// Mitsubishi GX Developer project: パレット取り外し   PLC: Q02

PROGRAM ALARM
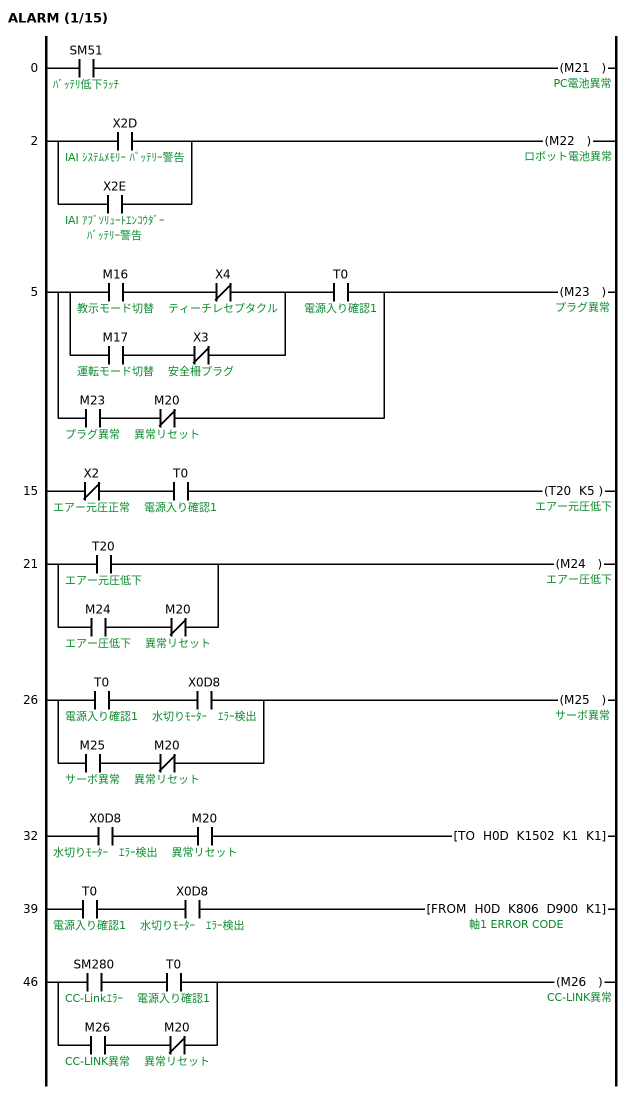
0     LD      SM51  ; ﾊﾞｯﾃﾘ低下ﾗｯﾁ
      OUT     M21  ; PC電池異常
2     LD      X2D  ; IAI ｼｽﾃﾑﾒﾓﾘｰ ﾊﾞｯﾃﾘｰ警告
      OR      X2E  ; IAI ｱﾌﾞｿﾘｭｰﾄｴﾝｺｳﾀﾞｰ ﾊﾞｯﾃﾘｰ警告
      OUT     M22  ; ロボット電池異常
5     LD      M16  ; 教示モード切替
      ANI     X4  ; ティーチレセプタクル
      LD      M17  ; 運転モード切替
      ANI     X3  ; 安全柵プラグ
      ORB
      AND     T0  ; 電源入り確認1
      LD      M23  ; プラグ異常
      ANI     M20  ; 異常リセット
      ORB
      OUT     M23  ; プラグ異常
15    LDI     X2  ; エアー元圧正常
      AND     T0  ; 電源入り確認1
      OUT     T20 K5  ; エアー元圧低下
21    LD      T20  ; エアー元圧低下
      LD      M24  ; エアー圧低下
      ANI     M20  ; 異常リセット
      ORB
      OUT     M24  ; エアー圧低下
26    LD      T0  ; 電源入り確認1
      AND     X0D8  ; 水切りﾓｰﾀｰ　ｴﾗｰ検出
      LD      M25  ; サーボ異常
      ANI     M20  ; 異常リセット
      ORB
      OUT     M25  ; サーボ異常
32    LD      X0D8  ; 水切りﾓｰﾀｰ　ｴﾗｰ検出
      AND     M20  ; 異常リセット
      TO      H0D K1502 K1 K1
39    LD      T0  ; 電源入り確認1
      AND     X0D8  ; 水切りﾓｰﾀｰ　ｴﾗｰ検出
      FROM    H0D K806 D900 K1  ; 軸1 ERROR CODE
46    LD      SM280  ; CC-Linkｴﾗｰ
      AND     T0  ; 電源入り確認1
      LD      M26  ; CC-LINK異常
      ANI     M20  ; 異常リセット
      ORB
      OUT     M26  ; CC-LINK異常
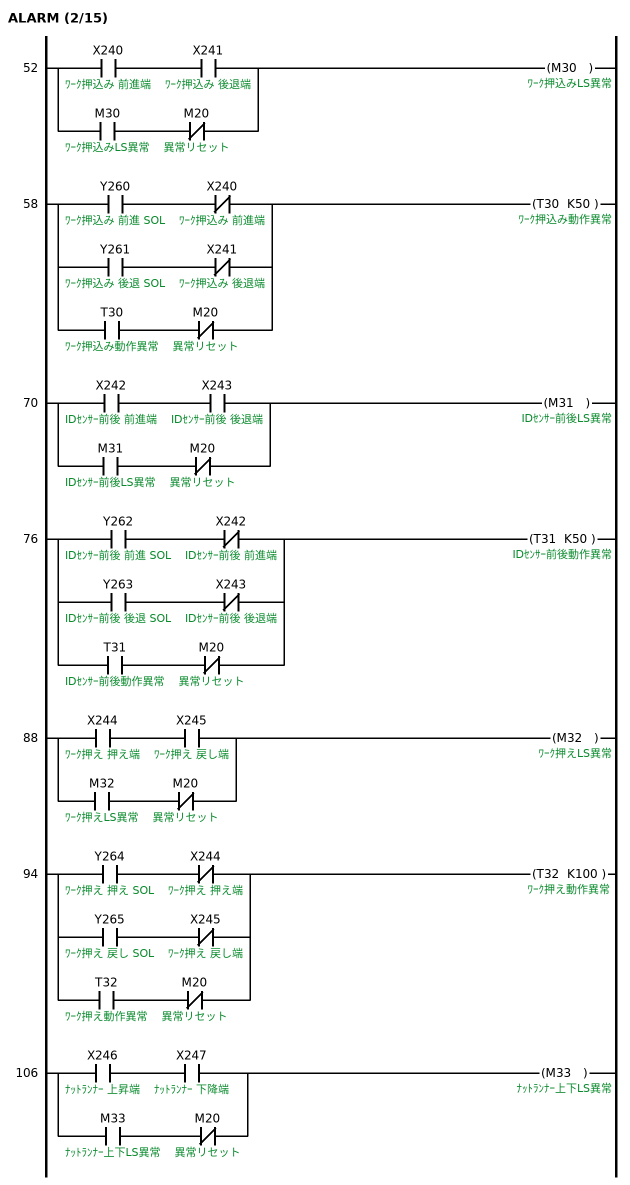
52    LD      X240  ; ﾜｰｸ押込み 前進端
      AND     X241  ; ﾜｰｸ押込み 後退端
      LD      M30  ; ﾜｰｸ押込みLS異常
      ANI     M20  ; 異常リセット
      ORB
      OUT     M30  ; ﾜｰｸ押込みLS異常
58    LD      Y260  ; ﾜｰｸ押込み 前進 SOL
      ANI     X240  ; ﾜｰｸ押込み 前進端
      LD      Y261  ; ﾜｰｸ押込み 後退 SOL
      ANI     X241  ; ﾜｰｸ押込み 後退端
      ORB
      LD      T30  ; ﾜｰｸ押込み動作異常
      ANI     M20  ; 異常リセット
      ORB
      OUT     T30 K50  ; ﾜｰｸ押込み動作異常
70    LD      X242  ; IDｾﾝｻｰ前後 前進端
      AND     X243  ; IDｾﾝｻｰ前後 後退端
      LD      M31  ; IDｾﾝｻｰ前後LS異常
      ANI     M20  ; 異常リセット
      ORB
      OUT     M31  ; IDｾﾝｻｰ前後LS異常
76    LD      Y262  ; IDｾﾝｻｰ前後 前進 SOL
      ANI     X242  ; IDｾﾝｻｰ前後 前進端
      LD      Y263  ; IDｾﾝｻｰ前後 後退 SOL
      ANI     X243  ; IDｾﾝｻｰ前後 後退端
      ORB
      LD      T31  ; IDｾﾝｻｰ前後動作異常
      ANI     M20  ; 異常リセット
      ORB
      OUT     T31 K50  ; IDｾﾝｻｰ前後動作異常
88    LD      X244  ; ﾜｰｸ押え 押え端
      AND     X245  ; ﾜｰｸ押え 戻し端
      LD      M32  ; ﾜｰｸ押えLS異常
      ANI     M20  ; 異常リセット
      ORB
      OUT     M32  ; ﾜｰｸ押えLS異常
94    LD      Y264  ; ﾜｰｸ押え 押え SOL
      ANI     X244  ; ﾜｰｸ押え 押え端
      LD      Y265  ; ﾜｰｸ押え 戻し SOL
      ANI     X245  ; ﾜｰｸ押え 戻し端
      ORB
      LD      T32  ; ﾜｰｸ押え動作異常
      ANI     M20  ; 異常リセット
      ORB
      OUT     T32 K100  ; ﾜｰｸ押え動作異常
106   LD      X246  ; ﾅｯﾄﾗﾝﾅｰ 上昇端
      AND     X247  ; ﾅｯﾄﾗﾝﾅｰ 下降端
      LD      M33  ; ﾅｯﾄﾗﾝﾅｰ上下LS異常
      ANI     M20  ; 異常リセット
      ORB
      OUT     M33  ; ﾅｯﾄﾗﾝﾅｰ上下LS異常
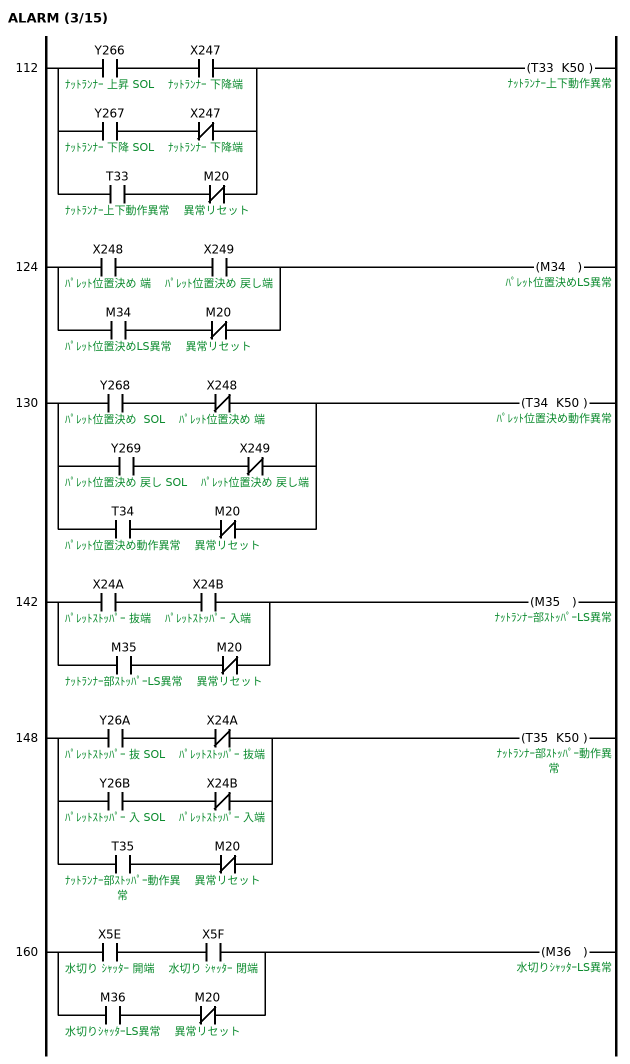
112   LD      Y266  ; ﾅｯﾄﾗﾝﾅｰ 上昇 SOL
      AND     X247  ; ﾅｯﾄﾗﾝﾅｰ 下降端
      LD      Y267  ; ﾅｯﾄﾗﾝﾅｰ 下降 SOL
      ANI     X247  ; ﾅｯﾄﾗﾝﾅｰ 下降端
      ORB
      LD      T33  ; ﾅｯﾄﾗﾝﾅｰ上下動作異常
      ANI     M20  ; 異常リセット
      ORB
      OUT     T33 K50  ; ﾅｯﾄﾗﾝﾅｰ上下動作異常
124   LD      X248  ; ﾊﾟﾚｯﾄ位置決め 端
      AND     X249  ; ﾊﾟﾚｯﾄ位置決め 戻し端
      LD      M34  ; ﾊﾟﾚｯﾄ位置決めLS異常
      ANI     M20  ; 異常リセット
      ORB
      OUT     M34  ; ﾊﾟﾚｯﾄ位置決めLS異常
130   LD      Y268  ; ﾊﾟﾚｯﾄ位置決め  SOL
      ANI     X248  ; ﾊﾟﾚｯﾄ位置決め 端
      LD      Y269  ; ﾊﾟﾚｯﾄ位置決め 戻し SOL
      ANI     X249  ; ﾊﾟﾚｯﾄ位置決め 戻し端
      ORB
      LD      T34  ; ﾊﾟﾚｯﾄ位置決め動作異常
      ANI     M20  ; 異常リセット
      ORB
      OUT     T34 K50  ; ﾊﾟﾚｯﾄ位置決め動作異常
142   LD      X24A  ; ﾊﾟﾚｯﾄｽﾄｯﾊﾟｰ 抜端
      AND     X24B  ; ﾊﾟﾚｯﾄｽﾄｯﾊﾟｰ 入端
      LD      M35  ; ﾅｯﾄﾗﾝﾅｰ部ｽﾄｯﾊﾟｰLS異常
      ANI     M20  ; 異常リセット
      ORB
      OUT     M35  ; ﾅｯﾄﾗﾝﾅｰ部ｽﾄｯﾊﾟｰLS異常
148   LD      Y26A  ; ﾊﾟﾚｯﾄｽﾄｯﾊﾟｰ 抜 SOL
      ANI     X24A  ; ﾊﾟﾚｯﾄｽﾄｯﾊﾟｰ 抜端
      LD      Y26B  ; ﾊﾟﾚｯﾄｽﾄｯﾊﾟｰ 入 SOL
      ANI     X24B  ; ﾊﾟﾚｯﾄｽﾄｯﾊﾟｰ 入端
      ORB
      LD      T35  ; ﾅｯﾄﾗﾝﾅｰ部ｽﾄｯﾊﾟｰ動作異常
      ANI     M20  ; 異常リセット
      ORB
      OUT     T35 K50  ; ﾅｯﾄﾗﾝﾅｰ部ｽﾄｯﾊﾟｰ動作異常
160   LD      X5E  ; 水切り ｼｬｯﾀｰ 開端
      AND     X5F  ; 水切り ｼｬｯﾀｰ 閉端
      LD      M36  ; 水切りｼｬｯﾀｰLS異常
      ANI     M20  ; 異常リセット
      ORB
      OUT     M36  ; 水切りｼｬｯﾀｰLS異常
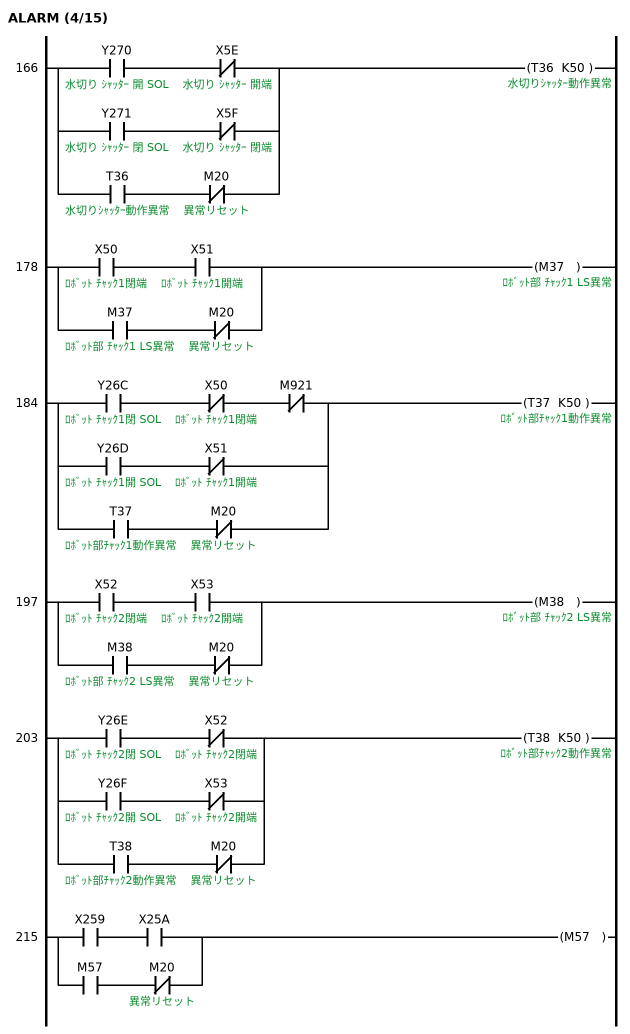
166   LD      Y270  ; 水切り ｼｬｯﾀｰ 開 SOL
      ANI     X5E  ; 水切り ｼｬｯﾀｰ 開端
      LD      Y271  ; 水切り ｼｬｯﾀｰ 閉 SOL
      ANI     X5F  ; 水切り ｼｬｯﾀｰ 閉端
      ORB
      LD      T36  ; 水切りｼｬｯﾀｰ動作異常
      ANI     M20  ; 異常リセット
      ORB
      OUT     T36 K50  ; 水切りｼｬｯﾀｰ動作異常
178   LD      X50  ; ﾛﾎﾞｯﾄ ﾁｬｯｸ1閉端
      AND     X51  ; ﾛﾎﾞｯﾄ ﾁｬｯｸ1開端
      LD      M37  ; ﾛﾎﾞｯﾄ部 ﾁｬｯｸ1 LS異常
      ANI     M20  ; 異常リセット
      ORB
      OUT     M37  ; ﾛﾎﾞｯﾄ部 ﾁｬｯｸ1 LS異常
184   LD      Y26C  ; ﾛﾎﾞｯﾄ ﾁｬｯｸ1閉 SOL
      ANI     X50  ; ﾛﾎﾞｯﾄ ﾁｬｯｸ1閉端
      ANI     M921
      LD      Y26D  ; ﾛﾎﾞｯﾄ ﾁｬｯｸ1開 SOL
      ANI     X51  ; ﾛﾎﾞｯﾄ ﾁｬｯｸ1開端
      ORB
      LD      T37  ; ﾛﾎﾞｯﾄ部ﾁｬｯｸ1動作異常
      ANI     M20  ; 異常リセット
      ORB
      OUT     T37 K50  ; ﾛﾎﾞｯﾄ部ﾁｬｯｸ1動作異常
197   LD      X52  ; ﾛﾎﾞｯﾄ ﾁｬｯｸ2閉端
      AND     X53  ; ﾛﾎﾞｯﾄ ﾁｬｯｸ2開端
      LD      M38  ; ﾛﾎﾞｯﾄ部 ﾁｬｯｸ2 LS異常
      ANI     M20  ; 異常リセット
      ORB
      OUT     M38  ; ﾛﾎﾞｯﾄ部 ﾁｬｯｸ2 LS異常
203   LD      Y26E  ; ﾛﾎﾞｯﾄ ﾁｬｯｸ2閉 SOL
      ANI     X52  ; ﾛﾎﾞｯﾄ ﾁｬｯｸ2閉端
      LD      Y26F  ; ﾛﾎﾞｯﾄ ﾁｬｯｸ2開 SOL
      ANI     X53  ; ﾛﾎﾞｯﾄ ﾁｬｯｸ2開端
      ORB
      LD      T38  ; ﾛﾎﾞｯﾄ部ﾁｬｯｸ2動作異常
      ANI     M20  ; 異常リセット
      ORB
      OUT     T38 K50  ; ﾛﾎﾞｯﾄ部ﾁｬｯｸ2動作異常
215   LD      X259
      AND     X25A
      LD      M57
      ANI     M20  ; 異常リセット
      ORB
      OUT     M57
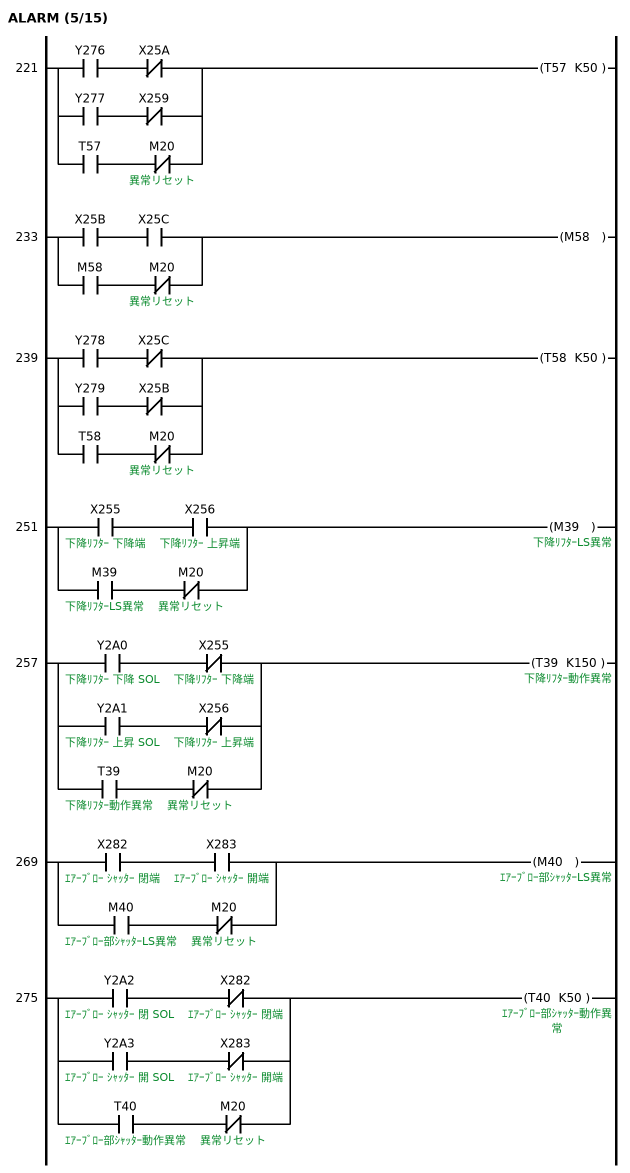
221   LD      Y276
      ANI     X25A
      LD      Y277
      ANI     X259
      ORB
      LD      T57
      ANI     M20  ; 異常リセット
      ORB
      OUT     T57 K50
233   LD      X25B
      AND     X25C
      LD      M58
      ANI     M20  ; 異常リセット
      ORB
      OUT     M58
239   LD      Y278
      ANI     X25C
      LD      Y279
      ANI     X25B
      ORB
      LD      T58
      ANI     M20  ; 異常リセット
      ORB
      OUT     T58 K50
251   LD      X255  ; 下降ﾘﾌﾀｰ 下降端
      AND     X256  ; 下降ﾘﾌﾀｰ 上昇端
      LD      M39  ; 下降ﾘﾌﾀｰLS異常
      ANI     M20  ; 異常リセット
      ORB
      OUT     M39  ; 下降ﾘﾌﾀｰLS異常
257   LD      Y2A0  ; 下降ﾘﾌﾀｰ 下降 SOL
      ANI     X255  ; 下降ﾘﾌﾀｰ 下降端
      LD      Y2A1  ; 下降ﾘﾌﾀｰ 上昇 SOL
      ANI     X256  ; 下降ﾘﾌﾀｰ 上昇端
      ORB
      LD      T39  ; 下降ﾘﾌﾀｰ動作異常
      ANI     M20  ; 異常リセット
      ORB
      OUT     T39 K150  ; 下降ﾘﾌﾀｰ動作異常
269   LD      X282  ; ｴｱｰﾌﾞﾛｰ ｼｬｯﾀｰ 閉端
      AND     X283  ; ｴｱｰﾌﾞﾛｰ ｼｬｯﾀｰ 開端
      LD      M40  ; ｴｱｰﾌﾞﾛｰ部ｼｬｯﾀｰLS異常
      ANI     M20  ; 異常リセット
      ORB
      OUT     M40  ; ｴｱｰﾌﾞﾛｰ部ｼｬｯﾀｰLS異常
275   LD      Y2A2  ; ｴｱｰﾌﾞﾛｰ ｼｬｯﾀｰ 閉 SOL
      ANI     X282  ; ｴｱｰﾌﾞﾛｰ ｼｬｯﾀｰ 閉端
      LD      Y2A3  ; ｴｱｰﾌﾞﾛｰ ｼｬｯﾀｰ 開 SOL
      ANI     X283  ; ｴｱｰﾌﾞﾛｰ ｼｬｯﾀｰ 開端
      ORB
      LD      T40  ; ｴｱｰﾌﾞﾛｰ部ｼｬｯﾀｰ動作異常
      ANI     M20  ; 異常リセット
      ORB
      OUT     T40 K50  ; ｴｱｰﾌﾞﾛｰ部ｼｬｯﾀｰ動作異常
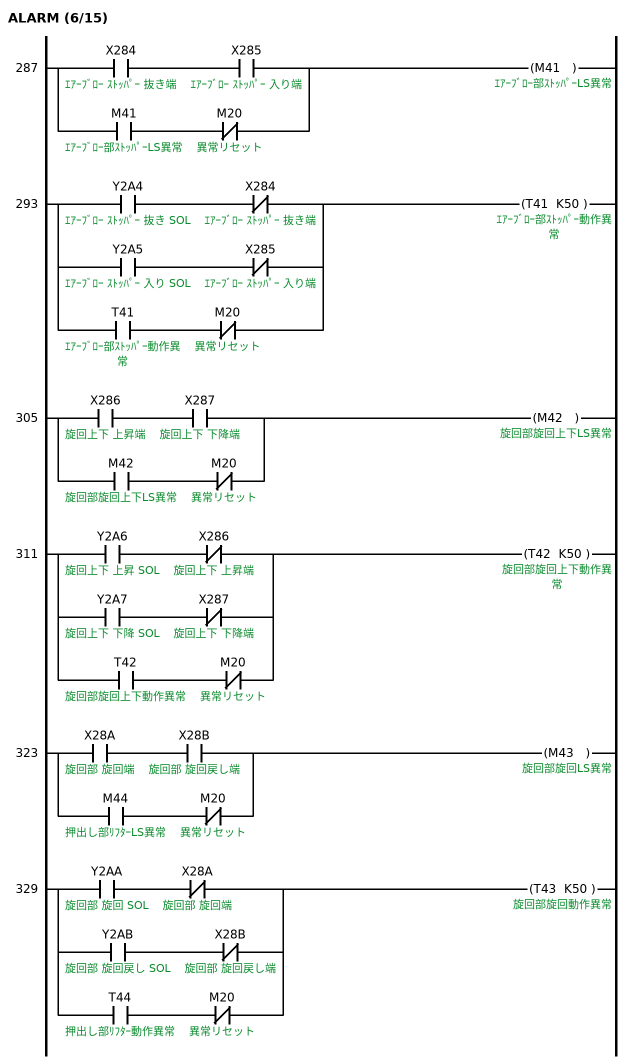
287   LD      X284  ; ｴｱｰﾌﾞﾛｰ ｽﾄｯﾊﾟｰ 抜き端
      AND     X285  ; ｴｱｰﾌﾞﾛｰ ｽﾄｯﾊﾟｰ 入り端
      LD      M41  ; ｴｱｰﾌﾞﾛｰ部ｽﾄｯﾊﾟｰLS異常
      ANI     M20  ; 異常リセット
      ORB
      OUT     M41  ; ｴｱｰﾌﾞﾛｰ部ｽﾄｯﾊﾟｰLS異常
293   LD      Y2A4  ; ｴｱｰﾌﾞﾛｰ ｽﾄｯﾊﾟｰ 抜き SOL
      ANI     X284  ; ｴｱｰﾌﾞﾛｰ ｽﾄｯﾊﾟｰ 抜き端
      LD      Y2A5  ; ｴｱｰﾌﾞﾛｰ ｽﾄｯﾊﾟｰ 入り SOL
      ANI     X285  ; ｴｱｰﾌﾞﾛｰ ｽﾄｯﾊﾟｰ 入り端
      ORB
      LD      T41  ; ｴｱｰﾌﾞﾛｰ部ｽﾄｯﾊﾟｰ動作異常
      ANI     M20  ; 異常リセット
      ORB
      OUT     T41 K50  ; ｴｱｰﾌﾞﾛｰ部ｽﾄｯﾊﾟｰ動作異常
305   LD      X286  ; 旋回上下 上昇端
      AND     X287  ; 旋回上下 下降端
      LD      M42  ; 旋回部旋回上下LS異常
      ANI     M20  ; 異常リセット
      ORB
      OUT     M42  ; 旋回部旋回上下LS異常
311   LD      Y2A6  ; 旋回上下 上昇 SOL
      ANI     X286  ; 旋回上下 上昇端
      LD      Y2A7  ; 旋回上下 下降 SOL
      ANI     X287  ; 旋回上下 下降端
      ORB
      LD      T42  ; 旋回部旋回上下動作異常
      ANI     M20  ; 異常リセット
      ORB
      OUT     T42 K50  ; 旋回部旋回上下動作異常
323   LD      X28A  ; 旋回部 旋回端
      AND     X28B  ; 旋回部 旋回戻し端
      LD      M44  ; 押出し部ﾘﾌﾀｰLS異常
      ANI     M20  ; 異常リセット
      ORB
      OUT     M43  ; 旋回部旋回LS異常
329   LD      Y2AA  ; 旋回部 旋回 SOL
      ANI     X28A  ; 旋回部 旋回端
      LD      Y2AB  ; 旋回部 旋回戻し SOL
      ANI     X28B  ; 旋回部 旋回戻し端
      ORB
      LD      T44  ; 押出し部ﾘﾌﾀｰ動作異常
      ANI     M20  ; 異常リセット
      ORB
      OUT     T43 K50  ; 旋回部旋回動作異常
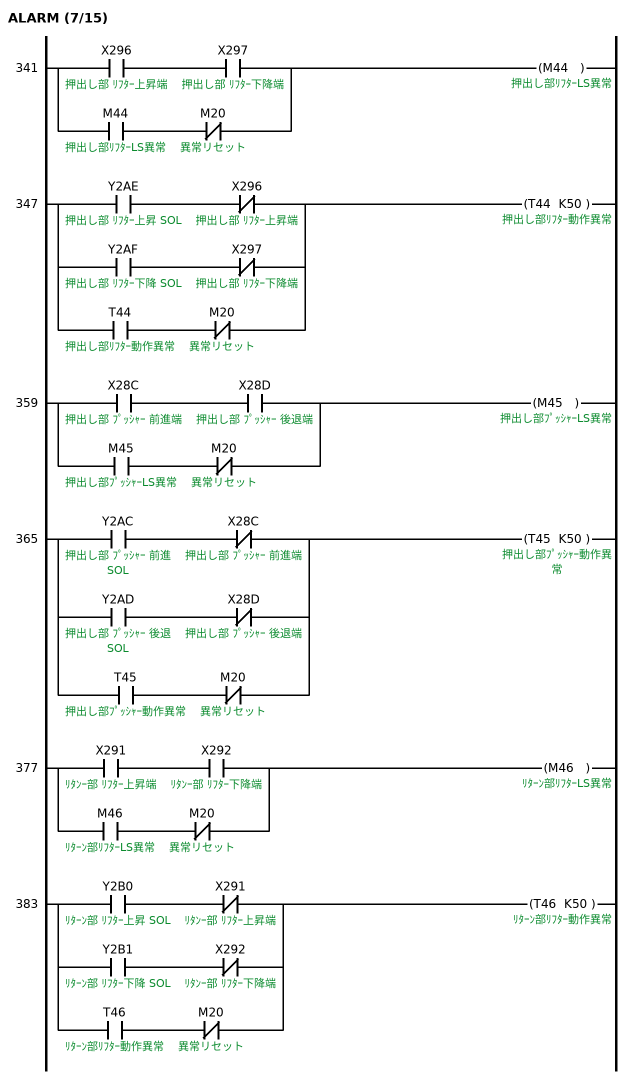
341   LD      X296  ; 押出し部 ﾘﾌﾀｰ上昇端
      AND     X297  ; 押出し部 ﾘﾌﾀｰ下降端
      LD      M44  ; 押出し部ﾘﾌﾀｰLS異常
      ANI     M20  ; 異常リセット
      ORB
      OUT     M44  ; 押出し部ﾘﾌﾀｰLS異常
347   LD      Y2AE  ; 押出し部 ﾘﾌﾀｰ上昇 SOL
      ANI     X296  ; 押出し部 ﾘﾌﾀｰ上昇端
      LD      Y2AF  ; 押出し部 ﾘﾌﾀｰ下降 SOL
      ANI     X297  ; 押出し部 ﾘﾌﾀｰ下降端
      ORB
      LD      T44  ; 押出し部ﾘﾌﾀｰ動作異常
      ANI     M20  ; 異常リセット
      ORB
      OUT     T44 K50  ; 押出し部ﾘﾌﾀｰ動作異常
359   LD      X28C  ; 押出し部 ﾌﾟｯｼｬｰ 前進端
      AND     X28D  ; 押出し部 ﾌﾟｯｼｬｰ 後退端
      LD      M45  ; 押出し部ﾌﾟｯｼｬｰLS異常
      ANI     M20  ; 異常リセット
      ORB
      OUT     M45  ; 押出し部ﾌﾟｯｼｬｰLS異常
365   LD      Y2AC  ; 押出し部 ﾌﾟｯｼｬｰ 前進 SOL
      ANI     X28C  ; 押出し部 ﾌﾟｯｼｬｰ 前進端
      LD      Y2AD  ; 押出し部 ﾌﾟｯｼｬｰ 後退 SOL
      ANI     X28D  ; 押出し部 ﾌﾟｯｼｬｰ 後退端
      ORB
      LD      T45  ; 押出し部ﾌﾟｯｼｬｰ動作異常
      ANI     M20  ; 異常リセット
      ORB
      OUT     T45 K50  ; 押出し部ﾌﾟｯｼｬｰ動作異常
377   LD      X291  ; ﾘﾀﾝｰ部 ﾘﾌﾀｰ上昇端
      AND     X292  ; ﾘﾀﾝｰ部 ﾘﾌﾀｰ下降端
      LD      M46  ; ﾘﾀｰﾝ部ﾘﾌﾀｰLS異常
      ANI     M20  ; 異常リセット
      ORB
      OUT     M46  ; ﾘﾀｰﾝ部ﾘﾌﾀｰLS異常
383   LD      Y2B0  ; ﾘﾀｰﾝ部 ﾘﾌﾀｰ上昇 SOL
      ANI     X291  ; ﾘﾀﾝｰ部 ﾘﾌﾀｰ上昇端
      LD      Y2B1  ; ﾘﾀｰﾝ部 ﾘﾌﾀｰ下降 SOL
      ANI     X292  ; ﾘﾀﾝｰ部 ﾘﾌﾀｰ下降端
      ORB
      LD      T46  ; ﾘﾀｰﾝ部ﾘﾌﾀｰ動作異常
      ANI     M20  ; 異常リセット
      ORB
      OUT     T46 K50  ; ﾘﾀｰﾝ部ﾘﾌﾀｰ動作異常
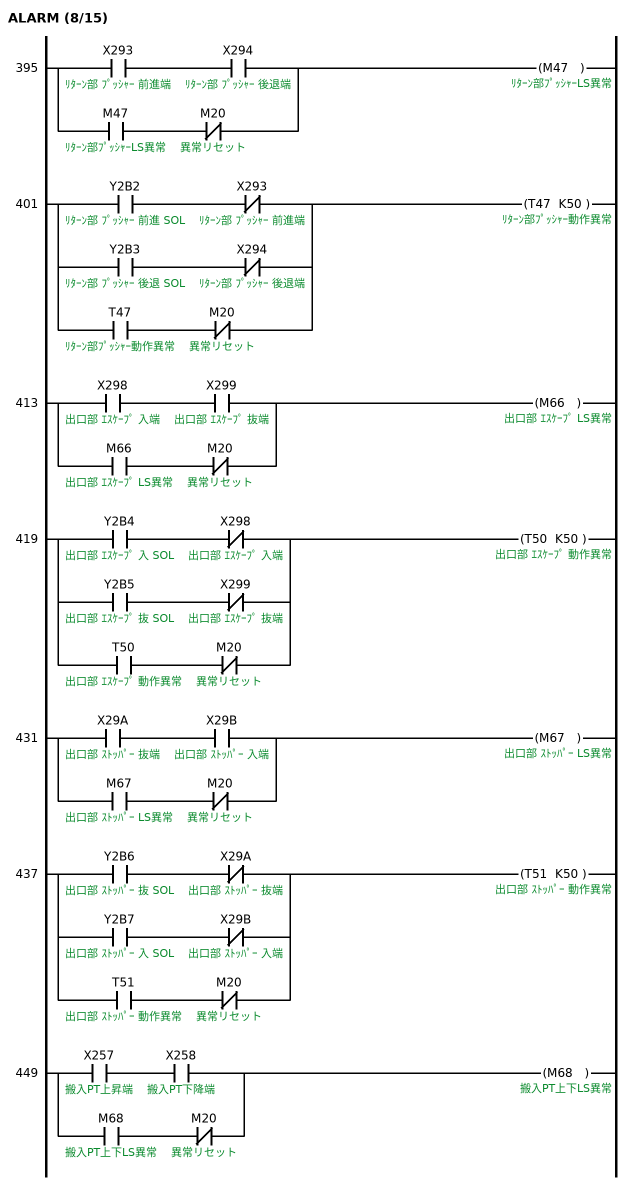
395   LD      X293  ; ﾘﾀｰﾝ部 ﾌﾟｯｼｬｰ 前進端
      AND     X294  ; ﾘﾀｰﾝ部 ﾌﾟｯｼｬｰ 後退端
      LD      M47  ; ﾘﾀｰﾝ部ﾌﾟｯｼｬｰLS異常
      ANI     M20  ; 異常リセット
      ORB
      OUT     M47  ; ﾘﾀｰﾝ部ﾌﾟｯｼｬｰLS異常
401   LD      Y2B2  ; ﾘﾀｰﾝ部 ﾌﾟｯｼｬｰ 前進 SOL
      ANI     X293  ; ﾘﾀｰﾝ部 ﾌﾟｯｼｬｰ 前進端
      LD      Y2B3  ; ﾘﾀｰﾝ部 ﾌﾟｯｼｬｰ 後退 SOL
      ANI     X294  ; ﾘﾀｰﾝ部 ﾌﾟｯｼｬｰ 後退端
      ORB
      LD      T47  ; ﾘﾀｰﾝ部ﾌﾟｯｼｬｰ動作異常
      ANI     M20  ; 異常リセット
      ORB
      OUT     T47 K50  ; ﾘﾀｰﾝ部ﾌﾟｯｼｬｰ動作異常
413   LD      X298  ; 出口部 ｴｽｹｰﾌﾟ 入端
      AND     X299  ; 出口部 ｴｽｹｰﾌﾟ 抜端
      LD      M66  ; 出口部 ｴｽｹｰﾌﾟ LS異常
      ANI     M20  ; 異常リセット
      ORB
      OUT     M66  ; 出口部 ｴｽｹｰﾌﾟ LS異常
419   LD      Y2B4  ; 出口部 ｴｽｹｰﾌﾟ 入 SOL
      ANI     X298  ; 出口部 ｴｽｹｰﾌﾟ 入端
      LD      Y2B5  ; 出口部 ｴｽｹｰﾌﾟ 抜 SOL
      ANI     X299  ; 出口部 ｴｽｹｰﾌﾟ 抜端
      ORB
      LD      T50  ; 出口部 ｴｽｹｰﾌﾟ 動作異常
      ANI     M20  ; 異常リセット
      ORB
      OUT     T50 K50  ; 出口部 ｴｽｹｰﾌﾟ 動作異常
431   LD      X29A  ; 出口部 ｽﾄｯﾊﾟｰ 抜端
      AND     X29B  ; 出口部 ｽﾄｯﾊﾟｰ 入端
      LD      M67  ; 出口部 ｽﾄｯﾊﾟｰ LS異常
      ANI     M20  ; 異常リセット
      ORB
      OUT     M67  ; 出口部 ｽﾄｯﾊﾟｰ LS異常
437   LD      Y2B6  ; 出口部 ｽﾄｯﾊﾟｰ 抜 SOL
      ANI     X29A  ; 出口部 ｽﾄｯﾊﾟｰ 抜端
      LD      Y2B7  ; 出口部 ｽﾄｯﾊﾟｰ 入 SOL
      ANI     X29B  ; 出口部 ｽﾄｯﾊﾟｰ 入端
      ORB
      LD      T51  ; 出口部 ｽﾄｯﾊﾟｰ 動作異常
      ANI     M20  ; 異常リセット
      ORB
      OUT     T51 K50  ; 出口部 ｽﾄｯﾊﾟｰ 動作異常
449   LD      X257  ; 搬入PT上昇端
      AND     X258  ; 搬入PT下降端
      LD      M68  ; 搬入PT上下LS異常
      ANI     M20  ; 異常リセット
      ORB
      OUT     M68  ; 搬入PT上下LS異常
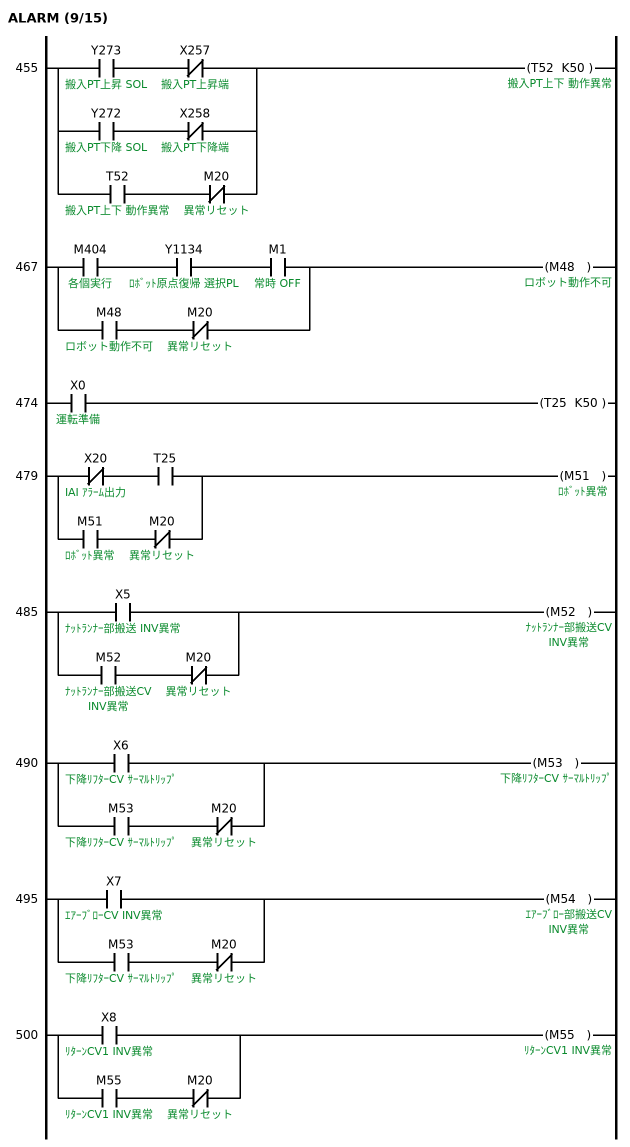
455   LD      Y273  ; 搬入PT上昇 SOL
      ANI     X257  ; 搬入PT上昇端
      LD      Y272  ; 搬入PT下降 SOL
      ANI     X258  ; 搬入PT下降端
      ORB
      LD      T52  ; 搬入PT上下 動作異常
      ANI     M20  ; 異常リセット
      ORB
      OUT     T52 K50  ; 搬入PT上下 動作異常
467   LD      M404  ; 各個実行
      AND     Y1134  ; ﾛﾎﾞｯﾄ原点復帰 選択PL
      AND     M1  ; 常時 OFF
      LD      M48  ; ロボット動作不可
      ANI     M20  ; 異常リセット
      ORB
      OUT     M48  ; ロボット動作不可
474   LD      X0  ; 運転準備
      OUT     T25 K50
479   LDI     X20  ; IAI ｱﾗｰﾑ出力
      AND     T25
      LD      M51  ; ﾛﾎﾞｯﾄ異常
      ANI     M20  ; 異常リセット
      ORB
      OUT     M51  ; ﾛﾎﾞｯﾄ異常
485   LD      X5  ; ﾅｯﾄﾗﾝﾅｰ部搬送 INV異常
      LD      M52  ; ﾅｯﾄﾗﾝﾅｰ部搬送CV INV異常
      ANI     M20  ; 異常リセット
      ORB
      OUT     M52  ; ﾅｯﾄﾗﾝﾅｰ部搬送CV INV異常
490   LD      X6  ; 下降ﾘﾌﾀｰCV ｻｰﾏﾙﾄﾘｯﾌﾟ
      LD      M53  ; 下降ﾘﾌﾀｰCV ｻｰﾏﾙﾄﾘｯﾌﾟ
      ANI     M20  ; 異常リセット
      ORB
      OUT     M53  ; 下降ﾘﾌﾀｰCV ｻｰﾏﾙﾄﾘｯﾌﾟ
495   LD      X7  ; ｴｱｰﾌﾞﾛｰCV INV異常
      LD      M53  ; 下降ﾘﾌﾀｰCV ｻｰﾏﾙﾄﾘｯﾌﾟ
      ANI     M20  ; 異常リセット
      ORB
      OUT     M54  ; ｴｱｰﾌﾞﾛｰ部搬送CV INV異常
500   LD      X8  ; ﾘﾀｰﾝCV1 INV異常
      LD      M55  ; ﾘﾀｰﾝCV1 INV異常
      ANI     M20  ; 異常リセット
      ORB
      OUT     M55  ; ﾘﾀｰﾝCV1 INV異常
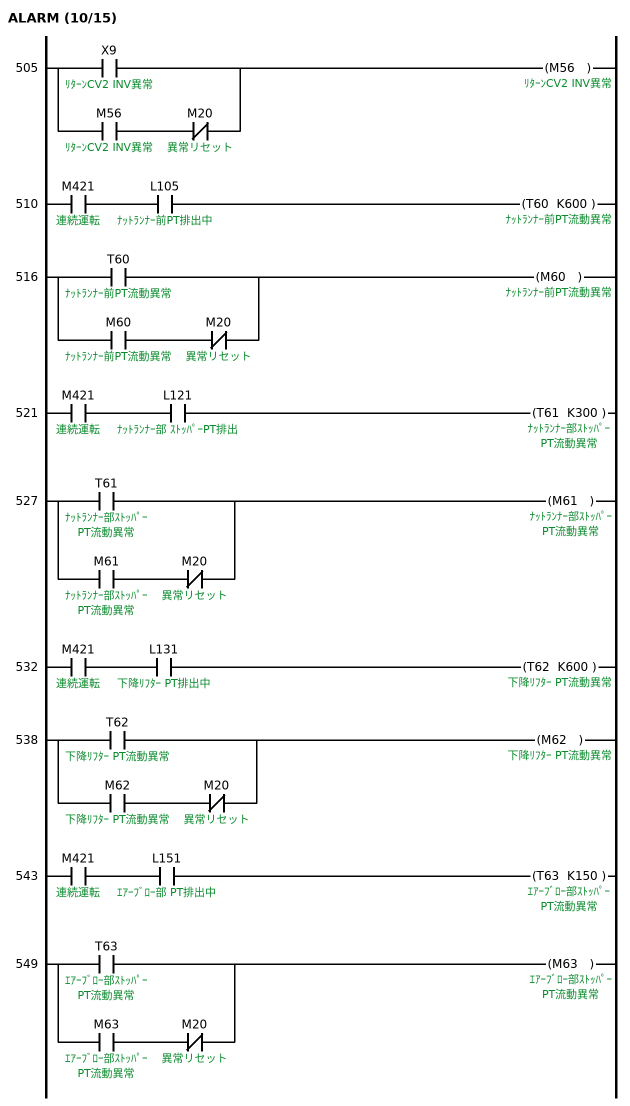
505   LD      X9  ; ﾘﾀｰﾝCV2 INV異常
      LD      M56  ; ﾘﾀｰﾝCV2 INV異常
      ANI     M20  ; 異常リセット
      ORB
      OUT     M56  ; ﾘﾀｰﾝCV2 INV異常
510   LD      M421  ; 連続運転
      AND     L105  ; ﾅｯﾄﾗﾝﾅｰ前PT排出中
      OUT     T60 K600  ; ﾅｯﾄﾗﾝﾅｰ前PT流動異常
516   LD      T60  ; ﾅｯﾄﾗﾝﾅｰ前PT流動異常
      LD      M60  ; ﾅｯﾄﾗﾝﾅｰ前PT流動異常
      ANI     M20  ; 異常リセット
      ORB
      OUT     M60  ; ﾅｯﾄﾗﾝﾅｰ前PT流動異常
521   LD      M421  ; 連続運転
      AND     L121  ; ﾅｯﾄﾗﾝﾅｰ部 ｽﾄｯﾊﾟｰPT排出
      OUT     T61 K300  ; ﾅｯﾄﾗﾝﾅｰ部ｽﾄｯﾊﾟｰ PT流動異常
527   LD      T61  ; ﾅｯﾄﾗﾝﾅｰ部ｽﾄｯﾊﾟｰ PT流動異常
      LD      M61  ; ﾅｯﾄﾗﾝﾅｰ部ｽﾄｯﾊﾟｰ PT流動異常
      ANI     M20  ; 異常リセット
      ORB
      OUT     M61  ; ﾅｯﾄﾗﾝﾅｰ部ｽﾄｯﾊﾟｰ PT流動異常
532   LD      M421  ; 連続運転
      AND     L131  ; 下降ﾘﾌﾀｰ PT排出中
      OUT     T62 K600  ; 下降ﾘﾌﾀｰ PT流動異常
538   LD      T62  ; 下降ﾘﾌﾀｰ PT流動異常
      LD      M62  ; 下降ﾘﾌﾀｰ PT流動異常
      ANI     M20  ; 異常リセット
      ORB
      OUT     M62  ; 下降ﾘﾌﾀｰ PT流動異常
543   LD      M421  ; 連続運転
      AND     L151  ; ｴｱｰﾌﾞﾛｰ部 PT排出中
      OUT     T63 K150  ; ｴｱｰﾌﾞﾛｰ部ｽﾄｯﾊﾟｰ PT流動異常
549   LD      T63  ; ｴｱｰﾌﾞﾛｰ部ｽﾄｯﾊﾟｰ PT流動異常
      LD      M63  ; ｴｱｰﾌﾞﾛｰ部ｽﾄｯﾊﾟｰ PT流動異常
      ANI     M20  ; 異常リセット
      ORB
      OUT     M63  ; ｴｱｰﾌﾞﾛｰ部ｽﾄｯﾊﾟｰ PT流動異常
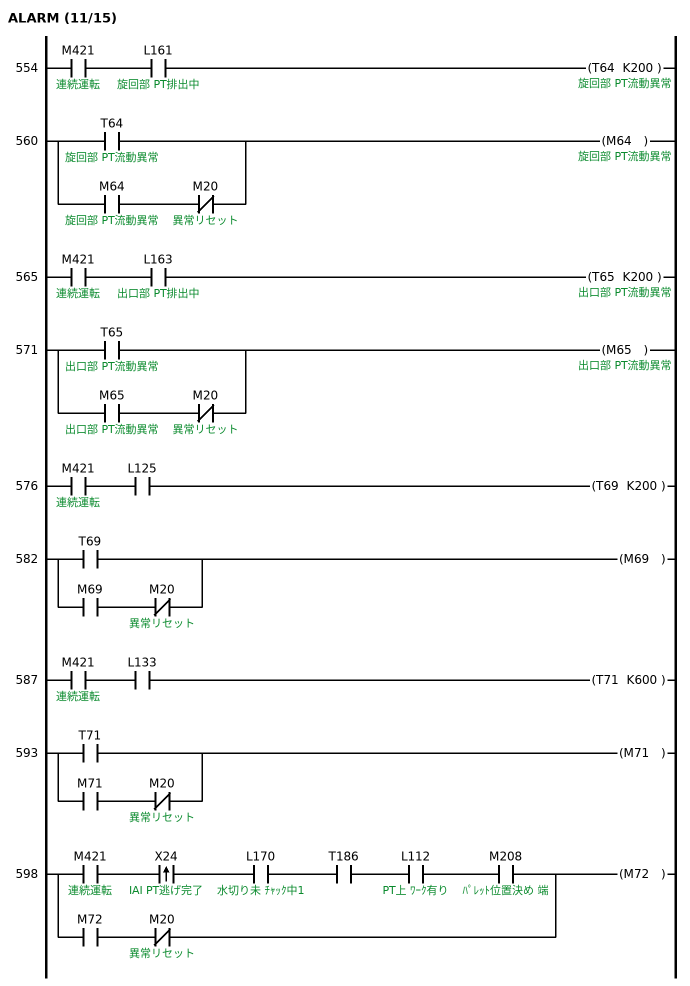
554   LD      M421  ; 連続運転
      AND     L161  ; 旋回部 PT排出中
      OUT     T64 K200  ; 旋回部 PT流動異常
560   LD      T64  ; 旋回部 PT流動異常
      LD      M64  ; 旋回部 PT流動異常
      ANI     M20  ; 異常リセット
      ORB
      OUT     M64  ; 旋回部 PT流動異常
565   LD      M421  ; 連続運転
      AND     L163  ; 出口部 PT排出中
      OUT     T65 K200  ; 出口部 PT流動異常
571   LD      T65  ; 出口部 PT流動異常
      LD      M65  ; 出口部 PT流動異常
      ANI     M20  ; 異常リセット
      ORB
      OUT     M65  ; 出口部 PT流動異常
576   LD      M421  ; 連続運転
      AND     L125
      OUT     T69 K200
582   LD      T69
      LD      M69
      ANI     M20  ; 異常リセット
      ORB
      OUT     M69
587   LD      M421  ; 連続運転
      AND     L133
      OUT     T71 K600
593   LD      T71
      LD      M71
      ANI     M20  ; 異常リセット
      ORB
      OUT     M71
598   LD      M421  ; 連続運転
      ANDP    X24  ; IAI PT逃げ完了
      AND     L170  ; 水切り未 ﾁｬｯｸ中1
      AND     T186
      AND     L112  ; PT上 ﾜｰｸ有り
      AND     M208  ; ﾊﾟﾚｯﾄ位置決め 端
      LD      M72
      ANI     M20  ; 異常リセット
      ORB
      OUT     M72
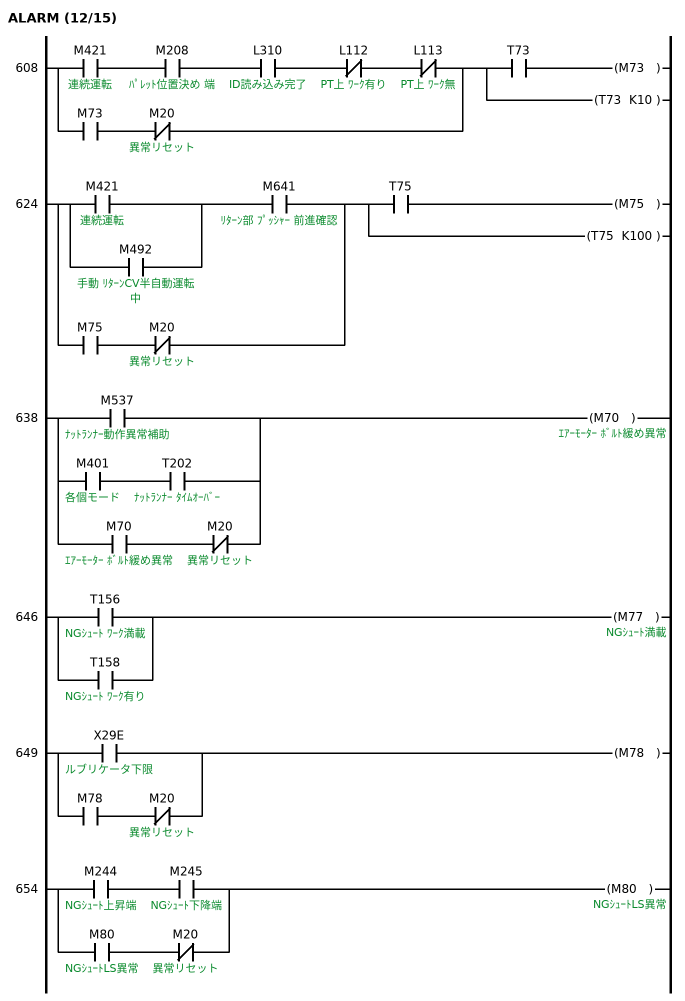
608   LD      M421  ; 連続運転
      AND     M208  ; ﾊﾟﾚｯﾄ位置決め 端
      AND     L310  ; ID読み込み完了
      ANI     L112  ; PT上 ﾜｰｸ有り
      ANI     L113  ; PT上 ﾜｰｸ無
      LD      M73
      ANI     M20  ; 異常リセット
      ORB
      MPS
      AND     T73
      OUT     M73
      MPP
      OUT     T73 K10
624   LD      M421  ; 連続運転
      OR      M492  ; 手動 ﾘﾀｰﾝCV半自動運転中
      AND     M641  ; ﾘﾀｰﾝ部 ﾌﾟｯｼｬｰ 前進確認
      LD      M75
      ANI     M20  ; 異常リセット
      ORB
      MPS
      AND     T75
      OUT     M75
      MPP
      OUT     T75 K100
638   LD      M537  ; ﾅｯﾄﾗﾝﾅｰ動作異常補助
      LD      M401  ; 各個モード
      AND     T202  ; ﾅｯﾄﾗﾝﾅｰ ﾀｲﾑｵｰﾊﾞｰ
      ORB
      LD      M70  ; ｴｱｰﾓｰﾀｰ ﾎﾞﾙﾄ緩め異常
      ANI     M20  ; 異常リセット
      ORB
      OUT     M70  ; ｴｱｰﾓｰﾀｰ ﾎﾞﾙﾄ緩め異常
646   LD      T156  ; NGｼｭｰﾄ ﾜｰｸ満載
      OR      T158  ; NGｼｭｰﾄ ﾜｰｸ有り
      OUT     M77  ; NGｼｭｰﾄ満載
649   LD      X29E  ; ルブリケータ下限
      LD      M78
      ANI     M20  ; 異常リセット
      ORB
      OUT     M78
654   LD      M244  ; NGｼｭｰﾄ上昇端
      AND     M245  ; NGｼｭｰﾄ下降端
      LD      M80  ; NGｼｭｰﾄLS異常
      ANI     M20  ; 異常リセット
      ORB
      OUT     M80  ; NGｼｭｰﾄLS異常
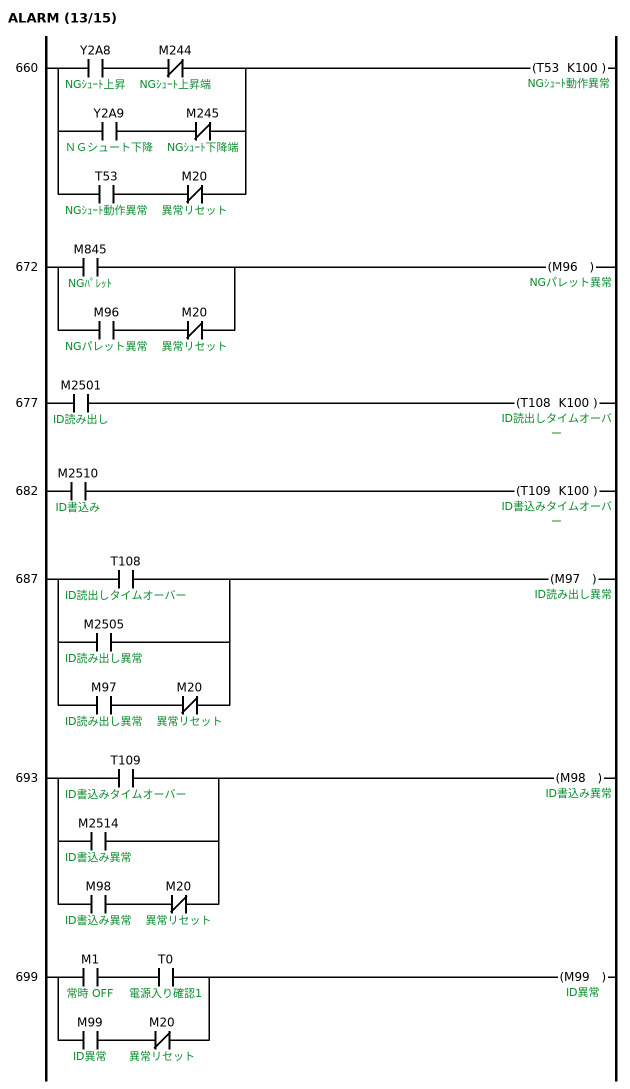
660   LD      Y2A8  ; NGｼｭｰﾄ上昇
      ANI     M244  ; NGｼｭｰﾄ上昇端
      LD      Y2A9  ; ＮＧシュート下降
      ANI     M245  ; NGｼｭｰﾄ下降端
      ORB
      LD      T53  ; NGｼｭｰﾄ動作異常
      ANI     M20  ; 異常リセット
      ORB
      OUT     T53 K100  ; NGｼｭｰﾄ動作異常
672   LD      M845  ; NGﾊﾟﾚｯﾄ
      LD      M96  ; NGパレット異常
      ANI     M20  ; 異常リセット
      ORB
      OUT     M96  ; NGパレット異常
677   LD      M2501  ; ID読み出し
      OUT     T108 K100  ; ID読出しタイムオーバー
682   LD      M2510  ; ID書込み
      OUT     T109 K100  ; ID書込みタイムオーバー
687   LD      T108  ; ID読出しタイムオーバー
      OR      M2505  ; ID読み出し異常
      LD      M97  ; ID読み出し異常
      ANI     M20  ; 異常リセット
      ORB
      OUT     M97  ; ID読み出し異常
693   LD      T109  ; ID書込みタイムオーバー
      OR      M2514  ; ID書込み異常
      LD      M98  ; ID書込み異常
      ANI     M20  ; 異常リセット
      ORB
      OUT     M98  ; ID書込み異常
699   LD      M1  ; 常時 OFF
      AND     T0  ; 電源入り確認1
      LD      M99  ; ID異常
      ANI     M20  ; 異常リセット
      ORB
      OUT     M99  ; ID異常
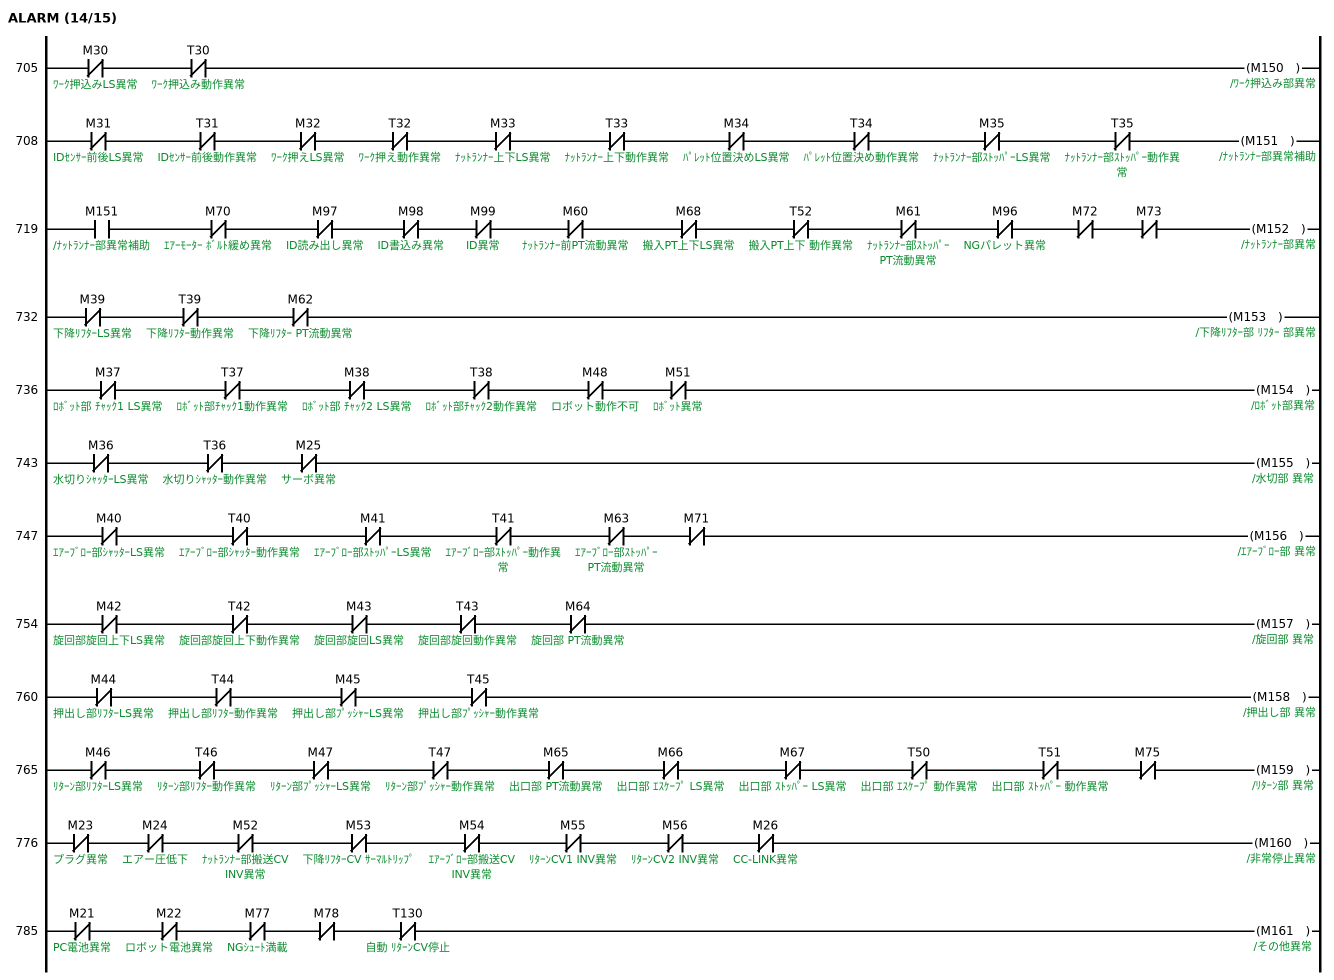
705   LDI     M30  ; ﾜｰｸ押込みLS異常
      ANI     T30  ; ﾜｰｸ押込み動作異常
      OUT     M150  ; /ﾜｰｸ押込み部異常
708   LDI     M31  ; IDｾﾝｻｰ前後LS異常
      ANI     T31  ; IDｾﾝｻｰ前後動作異常
      ANI     M32  ; ﾜｰｸ押えLS異常
      ANI     T32  ; ﾜｰｸ押え動作異常
      ANI     M33  ; ﾅｯﾄﾗﾝﾅｰ上下LS異常
      ANI     T33  ; ﾅｯﾄﾗﾝﾅｰ上下動作異常
      ANI     M34  ; ﾊﾟﾚｯﾄ位置決めLS異常
      ANI     T34  ; ﾊﾟﾚｯﾄ位置決め動作異常
      ANI     M35  ; ﾅｯﾄﾗﾝﾅｰ部ｽﾄｯﾊﾟｰLS異常
      ANI     T35  ; ﾅｯﾄﾗﾝﾅｰ部ｽﾄｯﾊﾟｰ動作異常
      OUT     M151  ; /ﾅｯﾄﾗﾝﾅｰ部異常補助
719   LD      M151  ; /ﾅｯﾄﾗﾝﾅｰ部異常補助
      ANI     M70  ; ｴｱｰﾓｰﾀｰ ﾎﾞﾙﾄ緩め異常
      ANI     M97  ; ID読み出し異常
      ANI     M98  ; ID書込み異常
      ANI     M99  ; ID異常
      ANI     M60  ; ﾅｯﾄﾗﾝﾅｰ前PT流動異常
      ANI     M68  ; 搬入PT上下LS異常
      ANI     T52  ; 搬入PT上下 動作異常
      ANI     M61  ; ﾅｯﾄﾗﾝﾅｰ部ｽﾄｯﾊﾟｰ PT流動異常
      ANI     M96  ; NGパレット異常
      ANI     M72
      ANI     M73
      OUT     M152  ; /ﾅｯﾄﾗﾝﾅｰ部異常
732   LDI     M39  ; 下降ﾘﾌﾀｰLS異常
      ANI     T39  ; 下降ﾘﾌﾀｰ動作異常
      ANI     M62  ; 下降ﾘﾌﾀｰ PT流動異常
      OUT     M153  ; /下降ﾘﾌﾀｰ部 ﾘﾌﾀｰ 部異常
736   LDI     M37  ; ﾛﾎﾞｯﾄ部 ﾁｬｯｸ1 LS異常
      ANI     T37  ; ﾛﾎﾞｯﾄ部ﾁｬｯｸ1動作異常
      ANI     M38  ; ﾛﾎﾞｯﾄ部 ﾁｬｯｸ2 LS異常
      ANI     T38  ; ﾛﾎﾞｯﾄ部ﾁｬｯｸ2動作異常
      ANI     M48  ; ロボット動作不可
      ANI     M51  ; ﾛﾎﾞｯﾄ異常
      OUT     M154  ; /ﾛﾎﾞｯﾄ部異常
743   LDI     M36  ; 水切りｼｬｯﾀｰLS異常
      ANI     T36  ; 水切りｼｬｯﾀｰ動作異常
      ANI     M25  ; サーボ異常
      OUT     M155  ; /水切部 異常
747   LDI     M40  ; ｴｱｰﾌﾞﾛｰ部ｼｬｯﾀｰLS異常
      ANI     T40  ; ｴｱｰﾌﾞﾛｰ部ｼｬｯﾀｰ動作異常
      ANI     M41  ; ｴｱｰﾌﾞﾛｰ部ｽﾄｯﾊﾟｰLS異常
      ANI     T41  ; ｴｱｰﾌﾞﾛｰ部ｽﾄｯﾊﾟｰ動作異常
      ANI     M63  ; ｴｱｰﾌﾞﾛｰ部ｽﾄｯﾊﾟｰ PT流動異常
      ANI     M71
      OUT     M156  ; /ｴｱｰﾌﾞﾛｰ部 異常
754   LDI     M42  ; 旋回部旋回上下LS異常
      ANI     T42  ; 旋回部旋回上下動作異常
      ANI     M43  ; 旋回部旋回LS異常
      ANI     T43  ; 旋回部旋回動作異常
      ANI     M64  ; 旋回部 PT流動異常
      OUT     M157  ; /旋回部 異常
760   LDI     M44  ; 押出し部ﾘﾌﾀｰLS異常
      ANI     T44  ; 押出し部ﾘﾌﾀｰ動作異常
      ANI     M45  ; 押出し部ﾌﾟｯｼｬｰLS異常
      ANI     T45  ; 押出し部ﾌﾟｯｼｬｰ動作異常
      OUT     M158  ; /押出し部 異常
765   LDI     M46  ; ﾘﾀｰﾝ部ﾘﾌﾀｰLS異常
      ANI     T46  ; ﾘﾀｰﾝ部ﾘﾌﾀｰ動作異常
      ANI     M47  ; ﾘﾀｰﾝ部ﾌﾟｯｼｬｰLS異常
      ANI     T47  ; ﾘﾀｰﾝ部ﾌﾟｯｼｬｰ動作異常
      ANI     M65  ; 出口部 PT流動異常
      ANI     M66  ; 出口部 ｴｽｹｰﾌﾟ LS異常
      ANI     M67  ; 出口部 ｽﾄｯﾊﾟｰ LS異常
      ANI     T50  ; 出口部 ｴｽｹｰﾌﾟ 動作異常
      ANI     T51  ; 出口部 ｽﾄｯﾊﾟｰ 動作異常
      ANI     M75
      OUT     M159  ; /ﾘﾀｰﾝ部 異常
776   LDI     M23  ; プラグ異常
      ANI     M24  ; エアー圧低下
      ANI     M52  ; ﾅｯﾄﾗﾝﾅｰ部搬送CV INV異常
      ANI     M53  ; 下降ﾘﾌﾀｰCV ｻｰﾏﾙﾄﾘｯﾌﾟ
      ANI     M54  ; ｴｱｰﾌﾞﾛｰ部搬送CV INV異常
      ANI     M55  ; ﾘﾀｰﾝCV1 INV異常
      ANI     M56  ; ﾘﾀｰﾝCV2 INV異常
      ANI     M26  ; CC-LINK異常
      OUT     M160  ; /非常停止異常
785   LDI     M21  ; PC電池異常
      ANI     M22  ; ロボット電池異常
      ANI     M77  ; NGｼｭｰﾄ満載
      ANI     M78
      ANI     T130  ; 自動 ﾘﾀｰﾝCV停止
      OUT     M161  ; /その他異常
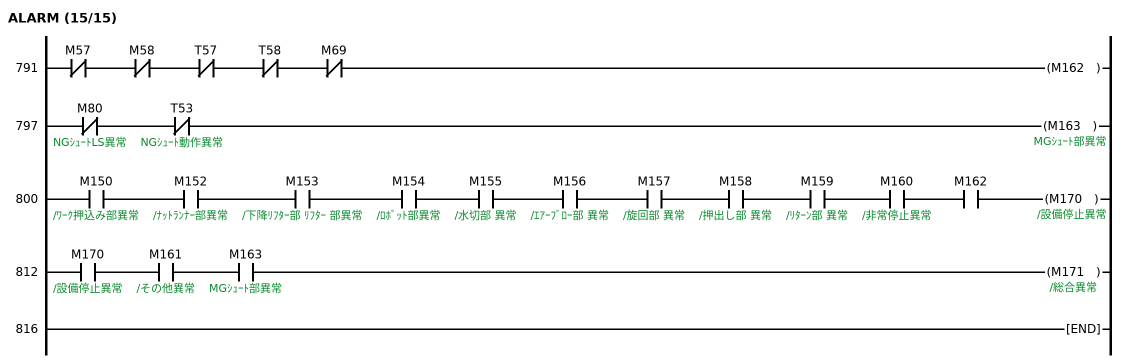
791   LDI     M57
      ANI     M58
      ANI     T57
      ANI     T58
      ANI     M69
      OUT     M162
797   LDI     M80  ; NGｼｭｰﾄLS異常
      ANI     T53  ; NGｼｭｰﾄ動作異常
      OUT     M163  ; MGｼｭｰﾄ部異常
800   LD      M150  ; /ﾜｰｸ押込み部異常
      AND     M152  ; /ﾅｯﾄﾗﾝﾅｰ部異常
      AND     M153  ; /下降ﾘﾌﾀｰ部 ﾘﾌﾀｰ 部異常
      AND     M154  ; /ﾛﾎﾞｯﾄ部異常
      AND     M155  ; /水切部 異常
      AND     M156  ; /ｴｱｰﾌﾞﾛｰ部 異常
      AND     M157  ; /旋回部 異常
      AND     M158  ; /押出し部 異常
      AND     M159  ; /ﾘﾀｰﾝ部 異常
      AND     M160  ; /非常停止異常
      AND     M162
      OUT     M170  ; /設備停止異常
812   LD      M170  ; /設備停止異常
      AND     M161  ; /その他異常
      AND     M163  ; MGｼｭｰﾄ部異常
      OUT     M171  ; /総合異常
816   END
END_PROGRAM
